FUNCTION_BLOCK T_RoboConnect_SetToolAnalogOutput_TimeoutFails EXTENDS T_UnitTestBase
VAR
  robot : I_RoboConnect;
  timeOutTimer : TON;
  targetAO : UINT;
  myTestState, prevState :
    (INIT,
    ARRANGE,
    ACT,
    ASSERT) := INIT;
  expected, actual : BOOL;
  counter : UINT;
  returnedTask : I_Task;
END_VAR

CASE myTestState OF
  INIT:
    StateChanged();
    myTestState := ARRANGE;

  ARRANGE:
    IF StateChanged() THEN
      expected := TRUE;
      robot.Connect();
    END_IF

    IF robot.Connected THEN
      myTestState := ACT;
    END_IF

  ACT:
    robot.SetDigitalOutput(targetAO,TRUE, task => returnedTask);
    myTestState := ASSERT;

  ASSERT:
    IF timeOutTimer.Q THEN
      actual := returnedTask.Timeout;
      assertion.AssertEquals_BOOL(expected, actual, 'actual := returnedTask.Timeout');
      TestFinished();
      myTestState := INIT;

    END_IF

END_CASE

robot.CyclicLogic();
timeOutTimer(IN := myTestState = ASSERT);

METHOD FB_init : BOOL
VAR_INPUT
  bInitRetains : BOOL; // if TRUE, the retain variables are initialized (warm start / cold start)
  bInCopyCode : BOOL; // if TRUE, the instance afterwards gets moved into the copy code (online change)
  TestSuite : tcl_SimpleUnitTestLibrary.I_TestSuite;
  robot : I_TcRobot;
  targetAo : UINT;
  timeout : TIME;
END_VAR
THIS^.robot := robot;
THIS^.timeoutTimer.PT := timeout;
THIS^.targetAo := targetAo;
END_METHOD

METHOD PRIVATE StateChanged : BOOL
IF  myTestState = prevState THEN
  RETURN;
END_IF

prevState := myTestState;
StateChanged := TRUE;
END_METHOD

METHOD WaitForCycles : BOOL
VAR_INPUT
  maxCount : UINT;
END_VAR
counter := counter + 1;

IF counter = maxCount THEN
  counter := 0;
  WaitForCycles := TRUE;
END_IF
END_METHOD

END_FUNCTION_BLOCK

(* stored: Version 1.1.0.1
   POU T_TcRobot_SetToolAnalogOutput_TimeoutFails: Id {b929a901-780e-4bde-9b67-f59b20783e7d}, SpecialFunc None
   Method FB_init: Id {c3bff287-6464-47dd-b53b-324fe67c7ea1}
   Method StateChanged: Id {93fbd318-a43a-4475-a870-f71e7e67eb56}
   Method WaitForCycles: Id {54539562-5336-4b69-a3c0-0c9fa33b8adc} *)
